{attribute 'qualified_only'}
VAR_GLOBAL
    {attribute 'TcLinkTo' := 'TIID^Device 2 (EtherCAT)^KF509 (PNOZ m ES EtherCAT)^SmPdoVariables^PNOZ_m_ES_EtherCAT__2_2__SM_3^TxPDO'}
    stPNOZEtherCATIn AT %I*: ST_PNOZEtherCATIn; //Raw EtherCAT input

    {attribute 'TcLinkTo' := 'TIID^Device 2 (EtherCAT)^KF509 (PNOZ m ES EtherCAT)^SmPdoVariables^PNOZ_m_ES_EtherCAT__2_2__SM_2^RxPDO'}
    stPNOZEtherCATOut AT %Q*: ST_PNOZEtherCATOut; //Raw EtherCAT output

    stPNOZEtherCATStatus: ST_PNOZEtherCATStatus; //Status struct for the PNOZ m ES EtherCAT, includes WcState and InfoData


    //Motion error registers from the Technosoft drives
    {attribute 'TcLinkTo' := '[1] := TIID^Device 2 (EtherCAT)^TA701 (iPOS8020 BX-CAT)^Transmit PDO 3 mapping parameters^Motion Error Register;
                              [2] := TIID^Device 2 (EtherCAT)^TA702 (iPOS8020 BX-CAT)^Transmit PDO 3 mapping parameters^Motion Error Register'}
    astTechnosoftMotionError AT %I*: ARRAY[1..cNBR_OF_TECHNOSOFT] OF ST_TechnosoftMotionError;

    {attribute 'TcLinkTo' := 'TIID^Device 2 (EtherCAT)^KF201 (EK1100)^KF208 (EL2014)^DIG Outputs^Channel 3^Output'}
    bSafetyAcknowledgeLED AT %Q*: BOOL;
END_VAR

VAR_GLOBAL CONSTANT
    cNBR_OF_SF: INT := 12;  //Virtual Output/Input bytes 04..15, each containing 8 bits
    cNBR_OF_TECHNOSOFT: INT := 2; //Number of Technosoft axises
END_VAR

(* stored: Version 1.1.0.1
   GVL GVL_SafetyIO: Id {a52cb188-5548-0f30-0b0b-19989305c2e3} *)
